(* Logix 5000 project; controller Amvex_Thorpe_Flowmeter vendor 1 type 14 code 106 rev 33.13; software revision 33.01; part 13 of 16 *)
(* tags used below, declared in another part *)
   Alicat0_ONS : BOOL;
   Alicat0DataInc : INT;
   Alicat1_ONS : BOOL;
   Alicat1DataInc : INT;
   Auto_Seq : SEQ;
   DonePallets : COUNTER;
   FAULT : DINT;
   FAULTED : DINT;
   MODE : MODE;
   RCD_ONS : BOOL;
   RESET : BOOL;
   Test : Connect;
   Alicat5LPM_Timeout : TIMER;
   Close_Rapid : Servo_Move;
   Close_Step : Servo_Move;
   CloseKnob : Servo_Move;
   FIRST_SCAN : BOOL;
   HMI : HMI_Temp;
   KB_DeBug : DINT;
   Load_PB_ONS : BOOL;
   MCP : MCP;
   Open : BOOL;
   Reject_Active : BOOL;
   Reject_Barcode : BOOL;
   Reject_CTR : COUNTER;
   Reject_Delay : BOOL;
   Reject_Pallet1_ONS : BOOL;
   Reject_Pallet_Bit : DINT;
   Safety_OK : BOOL;
   Test2_Rapid : Servo_Move;
   Test2_Step : Servo_Move;
   Test3_Rapid : Servo_Move;
   Test3_Step : Servo_Move;
   Test4_Rapid : Servo_Move;
   Test4_Step : Servo_Move;
   Test5_Rapid : Servo_Move;
   Test5_Step : Servo_Move;
   Test_Close : Servo_Move;
   Torque : DINT;
(* MCP_Main, continued *)

ROUTINE R04_CONV   (* ladder *)
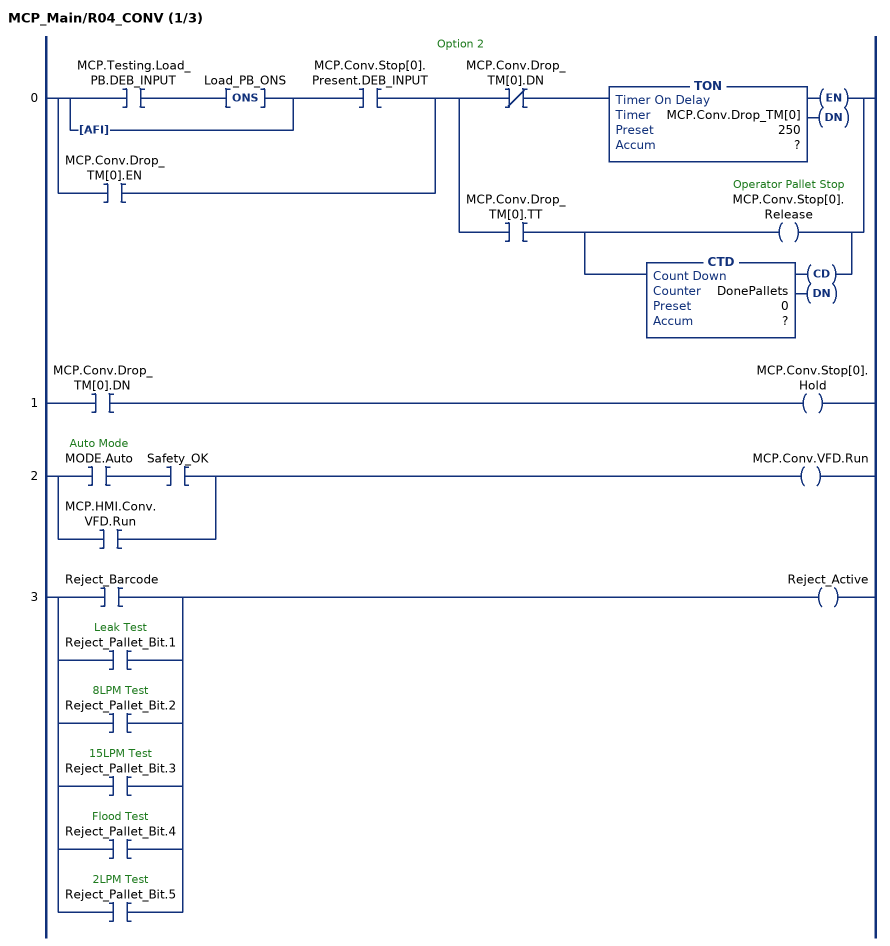
   // Option 2
   0: [[XIC(MCP.Testing.Load_PB.DEB_INPUT) ONS(Load_PB_ONS) ,AFI() ] XIC(MCP.Conv.Stop[0].Present.DEB_INPUT) ,XIC(MCP.Conv.Drop_TM[0].EN) ][XIO(MCP.Conv.Drop_TM[0].DN) TON(MCP.Conv.Drop_TM[0],?,?) ,XIC(MCP.Conv.Drop_TM[0].TT) [OTE(MCP.Conv.Stop[0].Release) ,CTD(DonePallets,?,?) ] ];
   1: XIC(MCP.Conv.Drop_TM[0].DN)OTE(MCP.Conv.Stop[0].Hold);
   2: [XIC(MODE.Auto) XIC(Safety_OK) ,XIC(MCP.HMI.Conv.VFD.Run) ]OTE(MCP.Conv.VFD.Run);
   3: [XIC(Reject_Barcode) ,XIC(Reject_Pallet_Bit.1) ,XIC(Reject_Pallet_Bit.2) ,XIC(Reject_Pallet_Bit.3) ,XIC(Reject_Pallet_Bit.4) ,XIC(Reject_Pallet_Bit.5) ]OTE(Reject_Active);
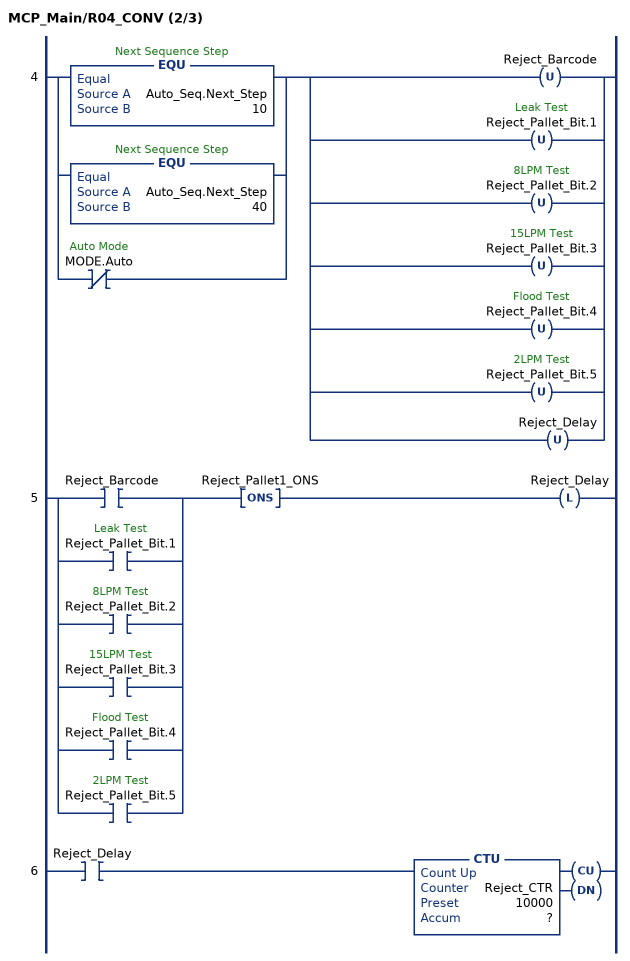
   4: [EQU(Auto_Seq.Next_Step,10) ,EQU(Auto_Seq.Next_Step,40) ,XIO(MODE.Auto) ][OTU(Reject_Barcode) ,OTU(Reject_Pallet_Bit.1) ,OTU(Reject_Pallet_Bit.2) ,OTU(Reject_Pallet_Bit.3) ,OTU(Reject_Pallet_Bit.4) ,OTU(Reject_Pallet_Bit.5) ,OTU(Reject_Delay) ];
   5: [XIC(Reject_Barcode) ,XIC(Reject_Pallet_Bit.1) ,XIC(Reject_Pallet_Bit.2) ,XIC(Reject_Pallet_Bit.3) ,XIC(Reject_Pallet_Bit.4) ,XIC(Reject_Pallet_Bit.5) ]ONS(Reject_Pallet1_ONS)OTL(Reject_Delay);
   6: XIC(Reject_Delay)CTU(Reject_CTR,?,?);
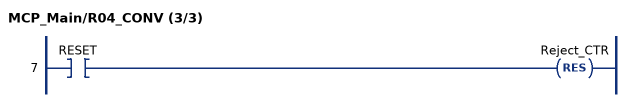
   7: XIC(RESET)RES(Reject_CTR);
END_ROUTINE

ROUTINE R05_FAULTS   (* ladder *)
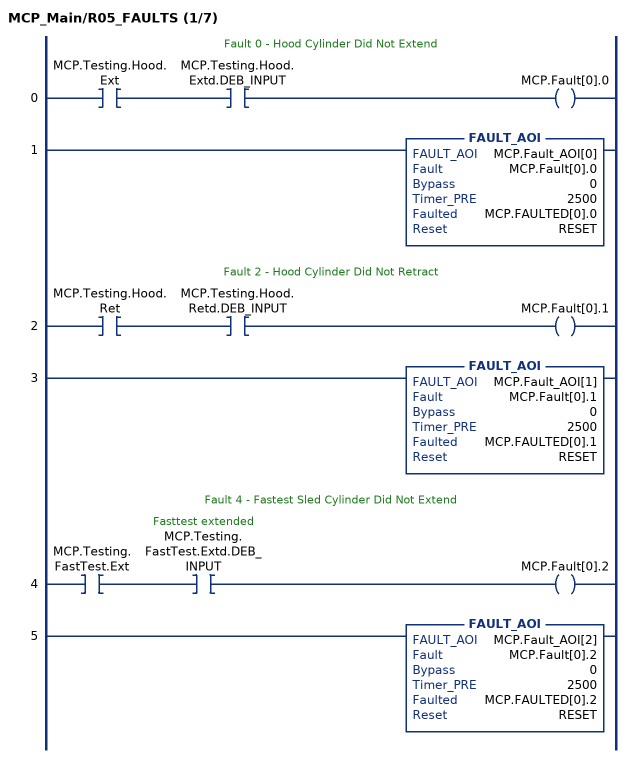
   // Fault 0 - Hood Cylinder Did Not Extend
   0: XIC(MCP.Testing.Hood.Ext)XIC(MCP.Testing.Hood.Extd.DEB_INPUT)OTE(MCP.Fault[0].0);
   1: FAULT_AOI(MCP.Fault_AOI[0],MCP.Fault[0].0,0,2500,MCP.FAULTED[0].0,RESET);
   // Fault 2 - Hood Cylinder Did Not Retract
   2: XIC(MCP.Testing.Hood.Ret)XIC(MCP.Testing.Hood.Retd.DEB_INPUT)OTE(MCP.Fault[0].1);
   3: FAULT_AOI(MCP.Fault_AOI[1],MCP.Fault[0].1,0,2500,MCP.FAULTED[0].1,RESET);
   // Fault 4 - Fastest Sled Cylinder Did Not Extend
   4: XIC(MCP.Testing.FastTest.Ext)XIC(MCP.Testing.FastTest.Extd.DEB_INPUT)OTE(MCP.Fault[0].2);
   5: FAULT_AOI(MCP.Fault_AOI[2],MCP.Fault[0].2,0,2500,MCP.FAULTED[0].2,RESET);
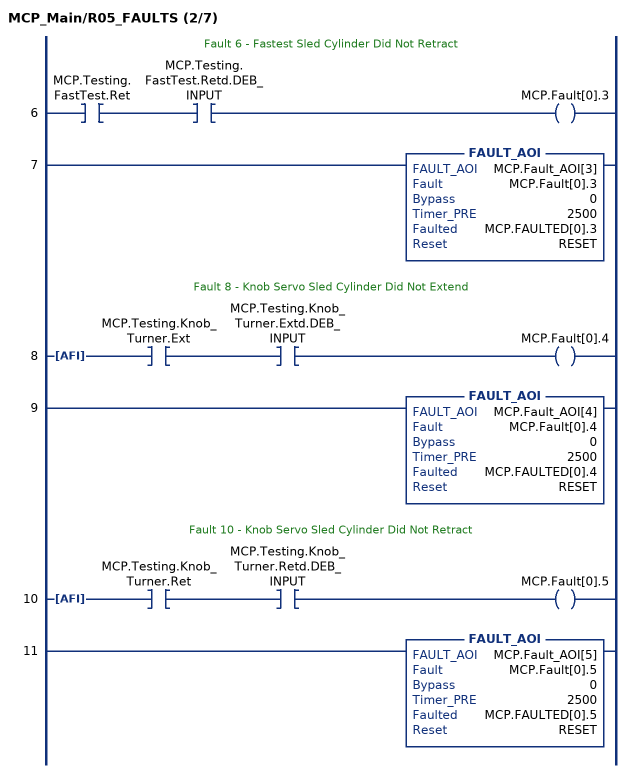
   // Fault 6 - Fastest Sled Cylinder Did Not Retract
   6: XIC(MCP.Testing.FastTest.Ret)XIC(MCP.Testing.FastTest.Retd.DEB_INPUT)OTE(MCP.Fault[0].3);
   7: FAULT_AOI(MCP.Fault_AOI[3],MCP.Fault[0].3,0,2500,MCP.FAULTED[0].3,RESET);
   // Fault 8 - Knob Servo Sled Cylinder Did Not Extend
   8: AFI()XIC(MCP.Testing.Knob_Turner.Ext)XIC(MCP.Testing.Knob_Turner.Extd.DEB_INPUT)OTE(MCP.Fault[0].4);
   9: FAULT_AOI(MCP.Fault_AOI[4],MCP.Fault[0].4,0,2500,MCP.FAULTED[0].4,RESET);
   // Fault 10 - Knob Servo Sled Cylinder Did Not Retract
   10: AFI()XIC(MCP.Testing.Knob_Turner.Ret)XIC(MCP.Testing.Knob_Turner.Retd.DEB_INPUT)OTE(MCP.Fault[0].5);
   11: FAULT_AOI(MCP.Fault_AOI[5],MCP.Fault[0].5,0,2500,MCP.FAULTED[0].5,RESET);
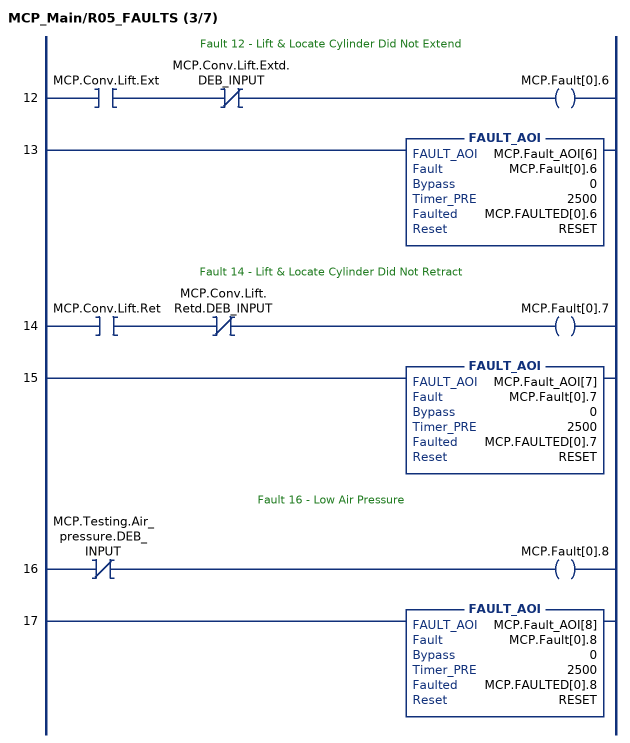
   // Fault 12 - Lift & Locate Cylinder Did Not Extend
   12: XIC(MCP.Conv.Lift.Ext)XIO(MCP.Conv.Lift.Extd.DEB_INPUT)OTE(MCP.Fault[0].6);
   13: FAULT_AOI(MCP.Fault_AOI[6],MCP.Fault[0].6,0,2500,MCP.FAULTED[0].6,RESET);
   // Fault 14 - Lift & Locate Cylinder Did Not Retract
   14: XIC(MCP.Conv.Lift.Ret)XIO(MCP.Conv.Lift.Retd.DEB_INPUT)OTE(MCP.Fault[0].7);
   15: FAULT_AOI(MCP.Fault_AOI[7],MCP.Fault[0].7,0,2500,MCP.FAULTED[0].7,RESET);
   // Fault 16 - Low Air Pressure
   16: XIO(MCP.Testing.Air_pressure.DEB_INPUT)OTE(MCP.Fault[0].8);
   17: FAULT_AOI(MCP.Fault_AOI[8],MCP.Fault[0].8,0,2500,MCP.FAULTED[0].8,RESET);
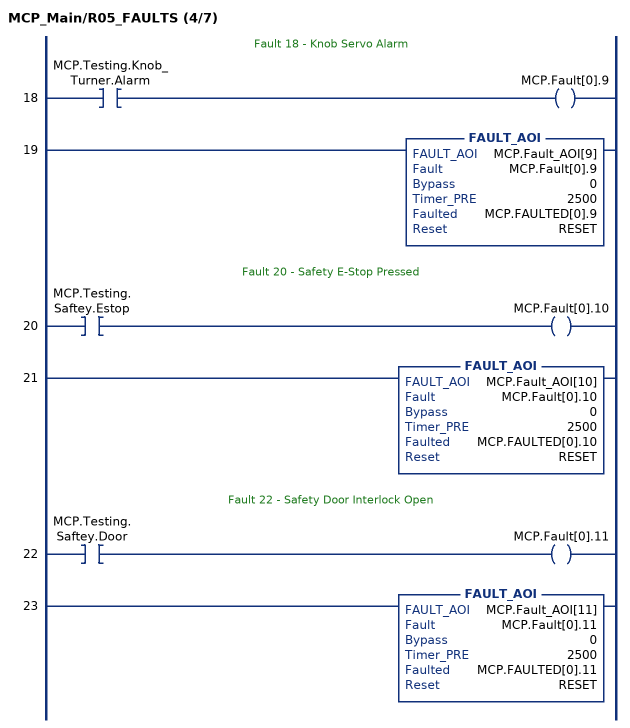
   // Fault 18 - Knob Servo Alarm
   18: XIC(MCP.Testing.Knob_Turner.Alarm)OTE(MCP.Fault[0].9);
   19: FAULT_AOI(MCP.Fault_AOI[9],MCP.Fault[0].9,0,2500,MCP.FAULTED[0].9,RESET);
   // Fault 20 - Safety E-Stop Pressed
   20: XIC(MCP.Testing.Saftey.Estop)OTE(MCP.Fault[0].10);
   21: FAULT_AOI(MCP.Fault_AOI[10],MCP.Fault[0].10,0,2500,MCP.FAULTED[0].10,RESET);
   // Fault 22 - Safety Door Interlock Open
   22: XIC(MCP.Testing.Saftey.Door)OTE(MCP.Fault[0].11);
   23: FAULT_AOI(MCP.Fault_AOI[11],MCP.Fault[0].11,0,2500,MCP.FAULTED[0].11,RESET);
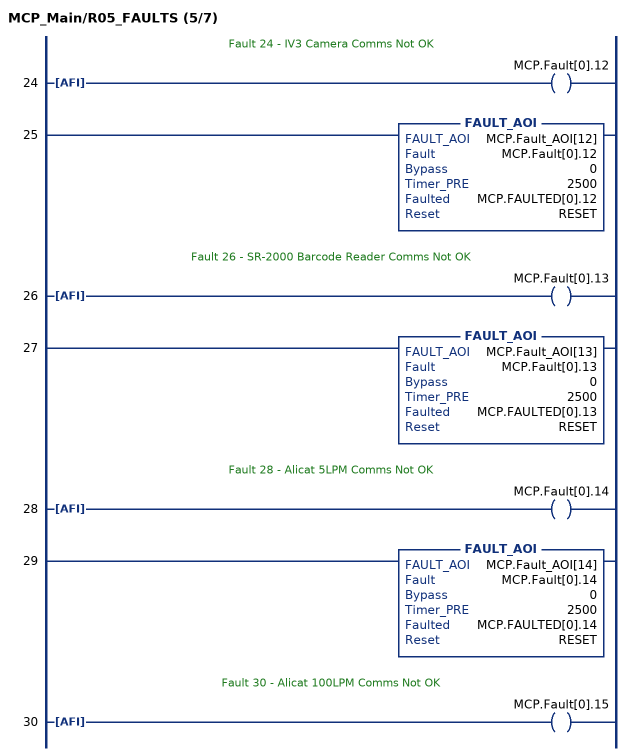
   // Fault 24 - IV3 Camera Comms Not OK
   24: AFI()OTE(MCP.Fault[0].12);
   25: FAULT_AOI(MCP.Fault_AOI[12],MCP.Fault[0].12,0,2500,MCP.FAULTED[0].12,RESET);
   // Fault 26 - SR-2000 Barcode Reader Comms Not OK
   26: AFI()OTE(MCP.Fault[0].13);
   27: FAULT_AOI(MCP.Fault_AOI[13],MCP.Fault[0].13,0,2500,MCP.FAULTED[0].13,RESET);
   // Fault 28 - Alicat 5LPM Comms Not OK
   28: AFI()OTE(MCP.Fault[0].14);
   29: FAULT_AOI(MCP.Fault_AOI[14],MCP.Fault[0].14,0,2500,MCP.FAULTED[0].14,RESET);
   // Fault 30 - Alicat 100LPM Comms Not OK
   30: AFI()OTE(MCP.Fault[0].15);
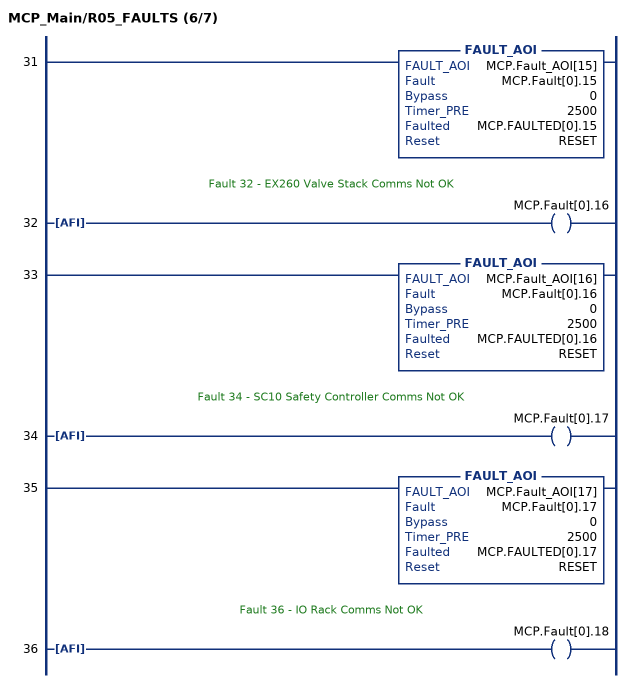
   31: FAULT_AOI(MCP.Fault_AOI[15],MCP.Fault[0].15,0,2500,MCP.FAULTED[0].15,RESET);
   // Fault 32 - EX260 Valve Stack Comms Not OK
   32: AFI()OTE(MCP.Fault[0].16);
   33: FAULT_AOI(MCP.Fault_AOI[16],MCP.Fault[0].16,0,2500,MCP.FAULTED[0].16,RESET);
   // Fault 34 - SC10 Safety Controller Comms Not OK
   34: AFI()OTE(MCP.Fault[0].17);
   35: FAULT_AOI(MCP.Fault_AOI[17],MCP.Fault[0].17,0,2500,MCP.FAULTED[0].17,RESET);
   // Fault 36 - IO Rack Comms Not OK
   36: AFI()OTE(MCP.Fault[0].18);
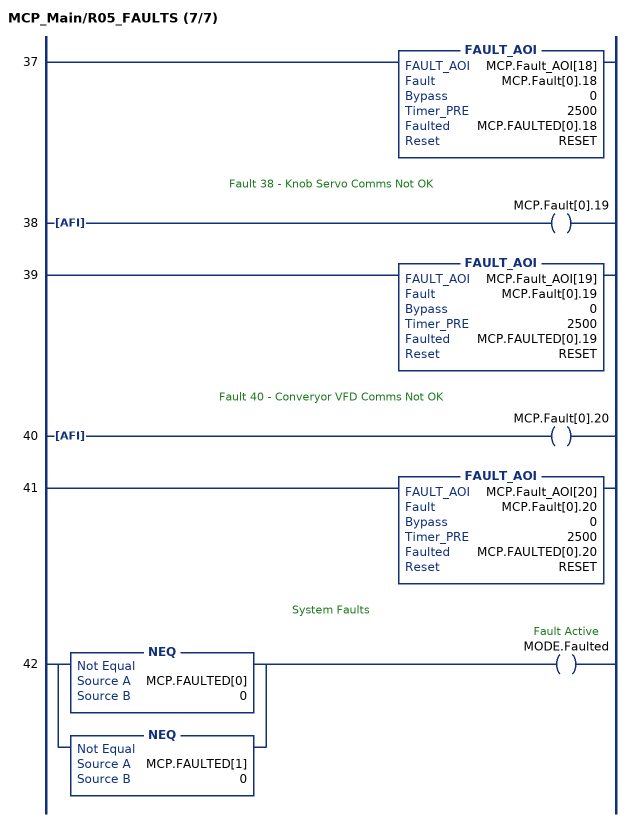
   37: FAULT_AOI(MCP.Fault_AOI[18],MCP.Fault[0].18,0,2500,MCP.FAULTED[0].18,RESET);
   // Fault 38 - Knob Servo Comms Not OK
   38: AFI()OTE(MCP.Fault[0].19);
   39: FAULT_AOI(MCP.Fault_AOI[19],MCP.Fault[0].19,0,2500,MCP.FAULTED[0].19,RESET);
   // Fault 40 - Converyor VFD Comms Not OK
   40: AFI()OTE(MCP.Fault[0].20);
   41: FAULT_AOI(MCP.Fault_AOI[20],MCP.Fault[0].20,0,2500,MCP.FAULTED[0].20,RESET);
   // System Faults
   42: [NEQ(MCP.FAULTED[0],0) ,NEQ(MCP.FAULTED[1],0) ]OTE(MODE.Faulted);
END_ROUTINE

ROUTINE R06_KNOB_TURNER   (* ladder *)
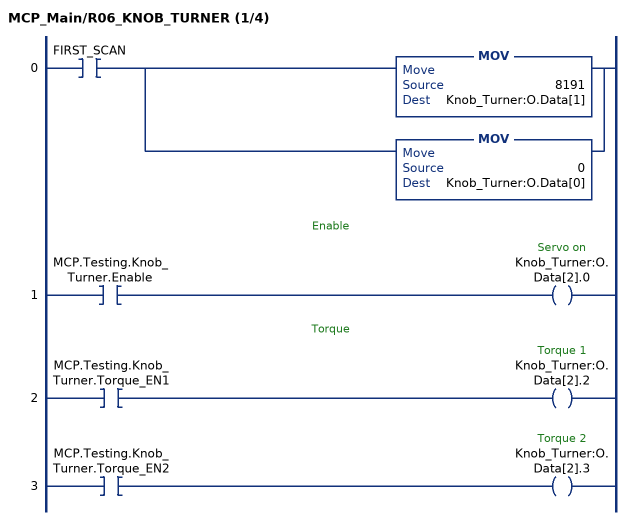
   0: XIC(FIRST_SCAN)[MOV(8191,Knob_Turner:O.Data[1]) ,MOV(0,Knob_Turner:O.Data[0]) ];
   // Enable
   1: XIC(MCP.Testing.Knob_Turner.Enable)OTE(Knob_Turner:O.Data[2].0);
   // Torque
   2: XIC(MCP.Testing.Knob_Turner.Torque_EN1)OTE(Knob_Turner:O.Data[2].2);
   3: XIC(MCP.Testing.Knob_Turner.Torque_EN2)OTE(Knob_Turner:O.Data[2].3);
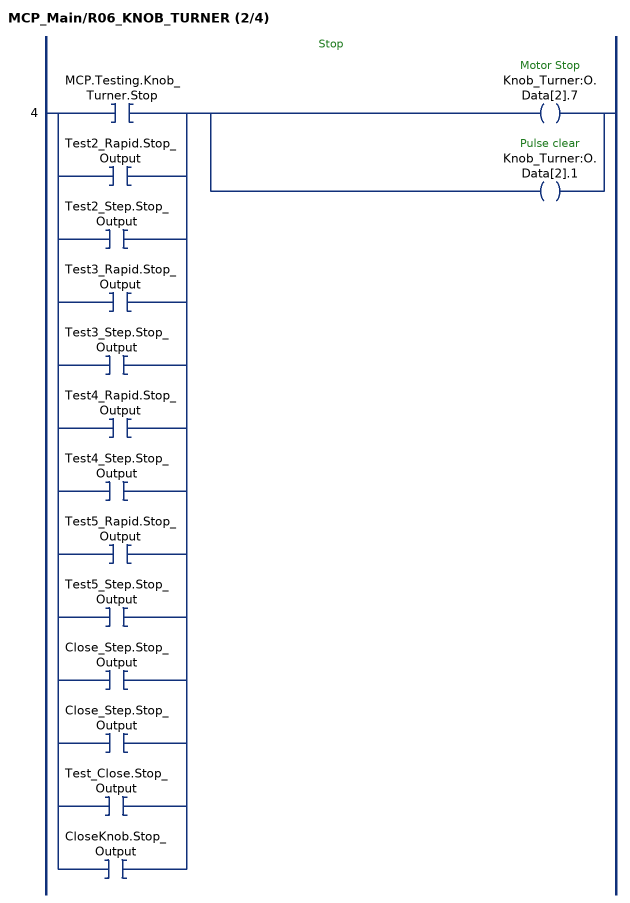
   // Stop
   4: [XIC(MCP.Testing.Knob_Turner.Stop) ,XIC(Test2_Rapid.Stop_Output) ,XIC(Test2_Step.Stop_Output) ,XIC(Test3_Rapid.Stop_Output) ,XIC(Test3_Step.Stop_Output) ,XIC(Test4_Rapid.Stop_Output) ,XIC(Test4_Step.Stop_Output) ,XIC(Test5_Rapid.Stop_Output) ,XIC(Test5_Step.Stop_Output) ,XIC(Close_Step.Stop_Output) ,XIC(Close_Step.Stop_Output) ,XIC(Test_Close.Stop_Output) ,XIC(CloseKnob.Stop_Output) ][OTE(Knob_Turner:O.Data[2].7) ,OTE(Knob_Turner:O.Data[2].1) ];
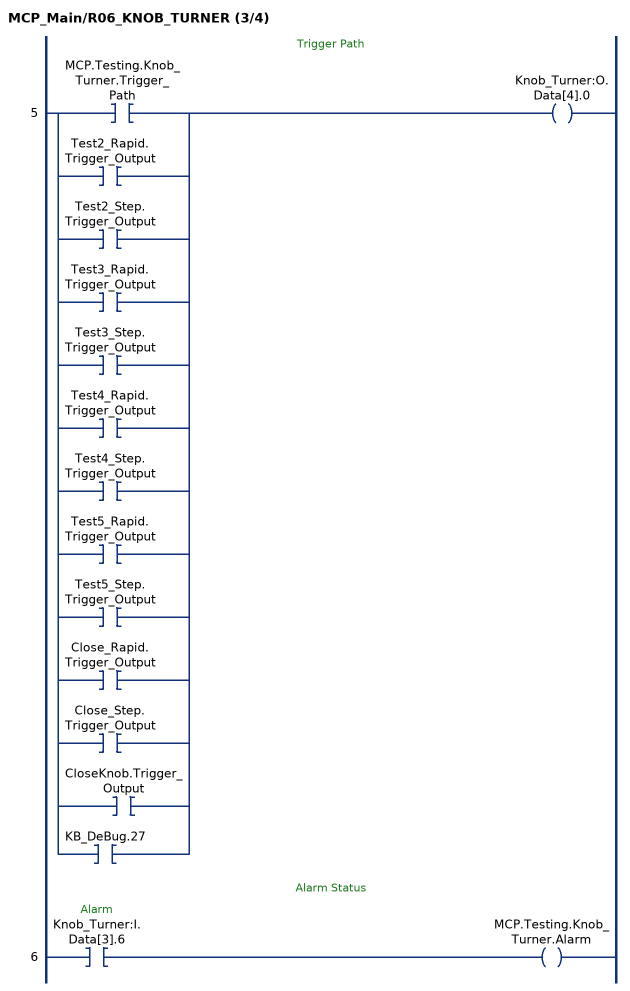
   // Trigger Path
   5: [XIC(MCP.Testing.Knob_Turner.Trigger_Path) ,XIC(Test2_Rapid.Trigger_Output) ,XIC(Test2_Step.Trigger_Output) ,XIC(Test3_Rapid.Trigger_Output) ,XIC(Test3_Step.Trigger_Output) ,XIC(Test4_Rapid.Trigger_Output) ,XIC(Test4_Step.Trigger_Output) ,XIC(Test5_Rapid.Trigger_Output) ,XIC(Test5_Step.Trigger_Output) ,XIC(Close_Rapid.Trigger_Output) ,XIC(Close_Step.Trigger_Output) ,XIC(CloseKnob.Trigger_Output) ,XIC(KB_DeBug.27) ]OTE(Knob_Turner:O.Data[4].0);
   // Alarm Status
   6: XIC(Knob_Turner:I.Data[3].6)OTE(MCP.Testing.Knob_Turner.Alarm);
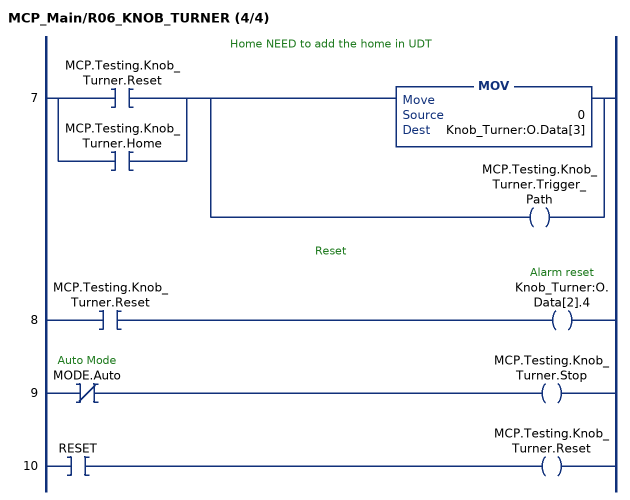
   // Home NEED to add the home in UDT
   7: [XIC(MCP.Testing.Knob_Turner.Reset) ,XIC(MCP.Testing.Knob_Turner.Home) ][MOV(0,Knob_Turner:O.Data[3]) ,OTE(MCP.Testing.Knob_Turner.Trigger_Path) ];
   // Reset
   8: XIC(MCP.Testing.Knob_Turner.Reset)OTE(Knob_Turner:O.Data[2].4);
   9: XIO(MODE.Auto)OTE(MCP.Testing.Knob_Turner.Stop);
   10: XIC(RESET)OTE(MCP.Testing.Knob_Turner.Reset);
END_ROUTINE

ROUTINE R07_SAFETY_CONTROLLER   (* ladder *)
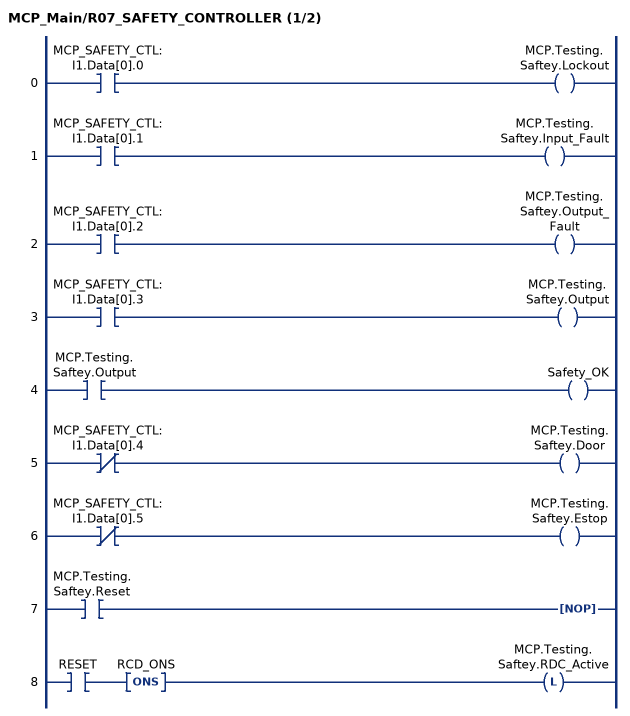
   0: XIC(MCP_SAFETY_CTL:I1.Data[0].0)OTE(MCP.Testing.Saftey.Lockout);
   1: XIC(MCP_SAFETY_CTL:I1.Data[0].1)OTE(MCP.Testing.Saftey.Input_Fault);
   2: XIC(MCP_SAFETY_CTL:I1.Data[0].2)OTE(MCP.Testing.Saftey.Output_Fault);
   3: XIC(MCP_SAFETY_CTL:I1.Data[0].3)OTE(MCP.Testing.Saftey.Output);
   4: XIC(MCP.Testing.Saftey.Output)OTE(Safety_OK);
   5: XIO(MCP_SAFETY_CTL:I1.Data[0].4)OTE(MCP.Testing.Saftey.Door);
   6: XIO(MCP_SAFETY_CTL:I1.Data[0].5)OTE(MCP.Testing.Saftey.Estop);
   7: XIC(MCP.Testing.Saftey.Reset)NOP();
   8: XIC(RESET)ONS(RCD_ONS)OTL(MCP.Testing.Saftey.RDC_Active);
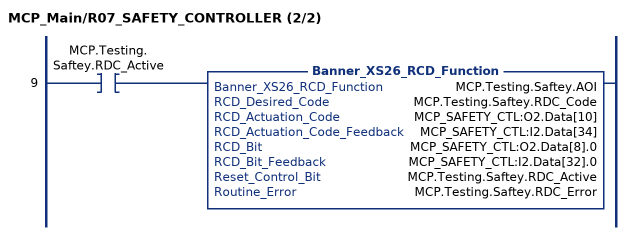
   9: XIC(MCP.Testing.Saftey.RDC_Active)Banner_XS26_RCD_Function(MCP.Testing.Saftey.AOI,MCP.Testing.Saftey.RDC_Code,MCP_SAFETY_CTL:O2.Data[10],MCP_SAFETY_CTL:I2.Data[34],MCP_SAFETY_CTL:O2.Data[8].0,MCP_SAFETY_CTL:I2.Data[32].0,MCP.Testing.Saftey.RDC_Active,MCP.Testing.Saftey.RDC_Error);
END_ROUTINE

ROUTINE R08_ALICATS   (* ladder *)
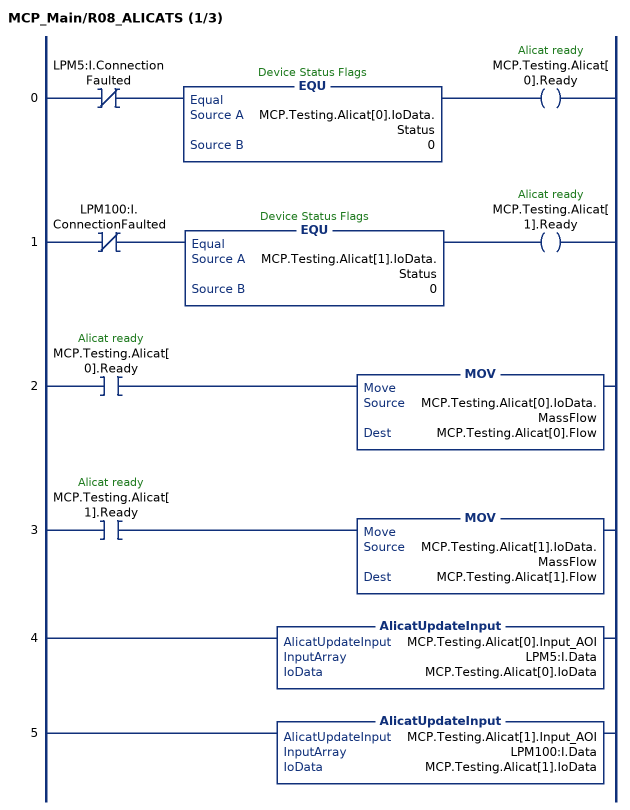
   0: XIO(LPM5:I.ConnectionFaulted)EQU(MCP.Testing.Alicat[0].IoData.Status,0)OTE(MCP.Testing.Alicat[0].Ready);
   1: XIO(LPM100:I.ConnectionFaulted)EQU(MCP.Testing.Alicat[1].IoData.Status,0)OTE(MCP.Testing.Alicat[1].Ready);
   2: XIC(MCP.Testing.Alicat[0].Ready)MOV(MCP.Testing.Alicat[0].IoData.MassFlow,MCP.Testing.Alicat[0].Flow);
   3: XIC(MCP.Testing.Alicat[1].Ready)MOV(MCP.Testing.Alicat[1].IoData.MassFlow,MCP.Testing.Alicat[1].Flow);
   4: AlicatUpdateInput(MCP.Testing.Alicat[0].Input_AOI,LPM5:I.Data,MCP.Testing.Alicat[0].IoData);
   5: AlicatUpdateInput(MCP.Testing.Alicat[1].Input_AOI,LPM100:I.Data,MCP.Testing.Alicat[1].IoData);
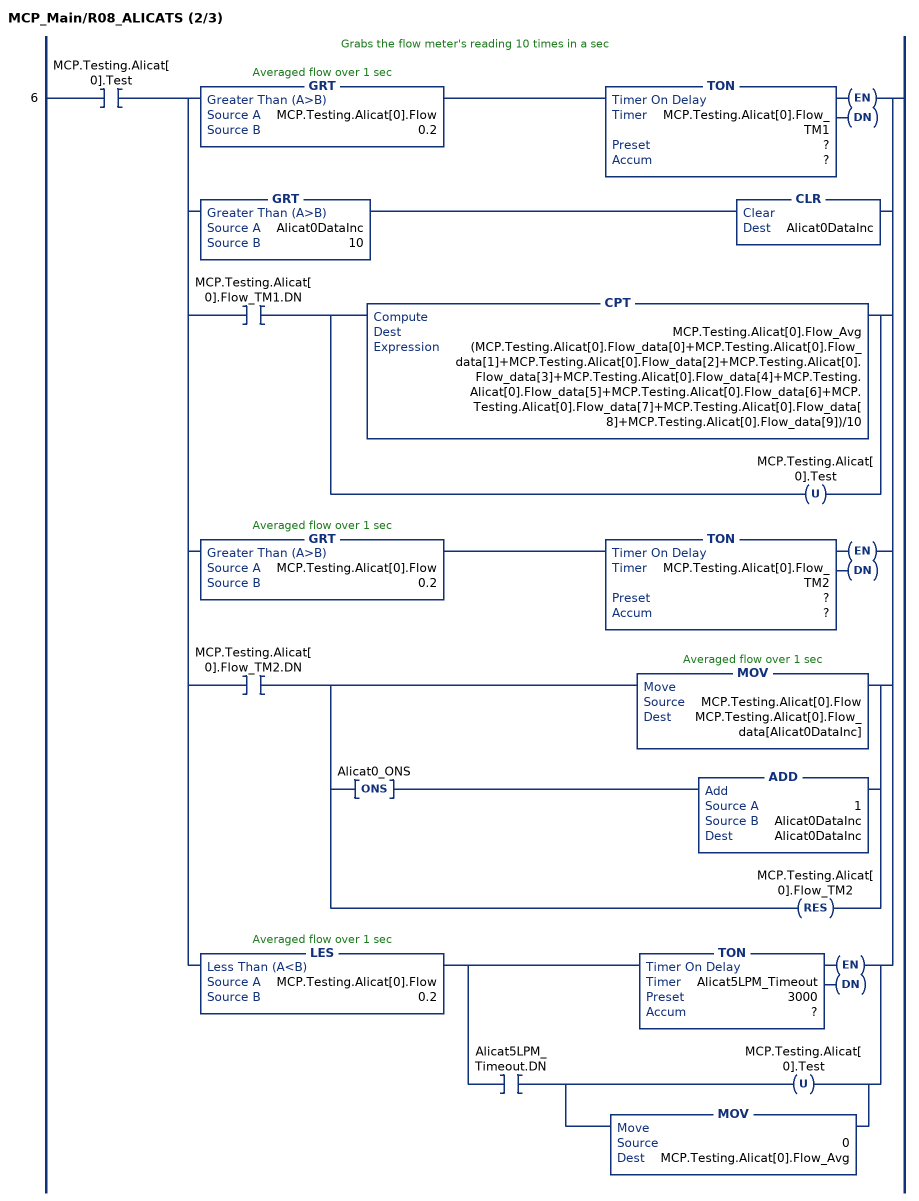
   // Grabs the flow meter's reading 10 times in a sec
   6: XIC(MCP.Testing.Alicat[0].Test)[[GRT(MCP.Testing.Alicat[0].Flow,0.2) TON(MCP.Testing.Alicat[0].Flow_TM1,?,?) ,GRT(Alicat0DataInc,10) CLR(Alicat0DataInc) ,XIC(MCP.Testing.Alicat[0].Flow_TM1.DN) [CPT(MCP.Testing.Alicat[0].Flow_Avg,(MCP.Testing.Alicat[0].Flow_data[0]+MCP.Testing.Alicat[0].Flow_data[1]+MCP.Testing.Alicat[0].Flow_data[2]+MCP.Testing.Alicat[0].Flow_data[3]+MCP.Testing.Alicat[0].Flow_data[4]+MCP.Testing.Alicat[0].Flow_data[5]+MCP.Testing.Alicat[0].Flow_data[6]+MCP.Testing.Alicat[0].Flow_data[7]+MCP.Testing.Alicat[0].Flow_data[8]+MCP.Testing.Alicat[0].Flow_data[9])/10) ,OTU(MCP.Testing.Alicat[0].Test) ] ,GRT(MCP.Testing.Alicat[0].Flow,0.2) TON(MCP.Testing.Alicat[0].Flow_TM2,?,?) ,XIC(MCP.Testing.Alicat[0].Flow_TM2.DN) [MOV(MCP.Testing.Alicat[0].Flow,MCP.Testing.Alicat[0].Flow_data[Alicat0DataInc]) ,ONS(Alicat0_ONS) ADD(1,Alicat0DataInc,Alicat0DataInc) ,RES(MCP.Testing.Alicat[0].Flow_TM2) ] ] ,LES(MCP.Testing.Alicat[0].Flow,0.2) [TON(Alicat5LPM_Timeout,?,?) ,XIC(Alicat5LPM_Timeout.DN) [OTU(MCP.Testing.Alicat[0].Test) ,MOV(0,MCP.Testing.Alicat[0].Flow_Avg) ] ] ];
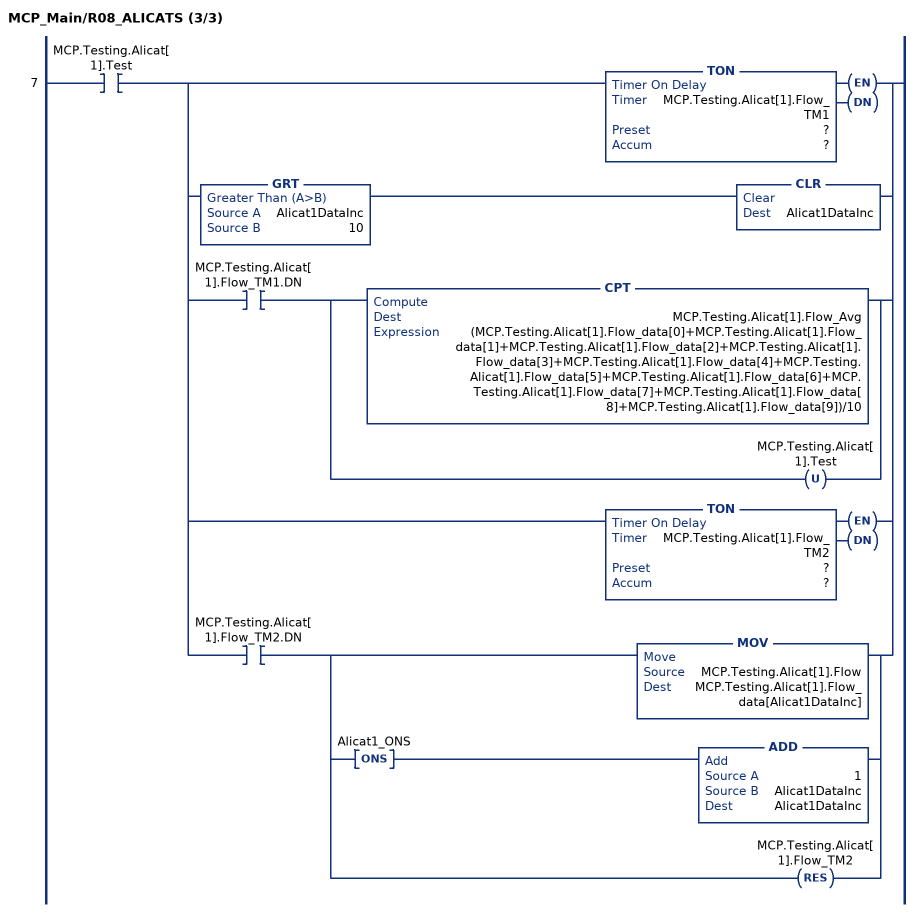
   7: XIC(MCP.Testing.Alicat[1].Test)[TON(MCP.Testing.Alicat[1].Flow_TM1,?,?) ,GRT(Alicat1DataInc,10) CLR(Alicat1DataInc) ,XIC(MCP.Testing.Alicat[1].Flow_TM1.DN) [CPT(MCP.Testing.Alicat[1].Flow_Avg,(MCP.Testing.Alicat[1].Flow_data[0]+MCP.Testing.Alicat[1].Flow_data[1]+MCP.Testing.Alicat[1].Flow_data[2]+MCP.Testing.Alicat[1].Flow_data[3]+MCP.Testing.Alicat[1].Flow_data[4]+MCP.Testing.Alicat[1].Flow_data[5]+MCP.Testing.Alicat[1].Flow_data[6]+MCP.Testing.Alicat[1].Flow_data[7]+MCP.Testing.Alicat[1].Flow_data[8]+MCP.Testing.Alicat[1].Flow_data[9])/10) ,OTU(MCP.Testing.Alicat[1].Test) ] ,TON(MCP.Testing.Alicat[1].Flow_TM2,?,?) ,XIC(MCP.Testing.Alicat[1].Flow_TM2.DN) [MOV(MCP.Testing.Alicat[1].Flow,MCP.Testing.Alicat[1].Flow_data[Alicat1DataInc]) ,ONS(Alicat1_ONS) ADD(1,Alicat1DataInc,Alicat1DataInc) ,RES(MCP.Testing.Alicat[1].Flow_TM2) ] ];
END_ROUTINE
